// TIA Portal V17 export
// export: Created 2024-08-29T18:23:45.4451093Z, ExportSetting WithDefaults, DisplayName Totally Integrated Automation Portal, DisplayVersion V17 Update 7, DisplayName TIA Portal Openness, DisplayVersion V17 Update 7, DisplayName TIA Portal Version Control Interface, DisplayVersion V17, DisplayName SINAMICS Startdrive Advanced, DisplayVersion V17 SP2, DisplayName SINAMICS Startdrive G110M, G120, G120C, G120D, G120P, G115D, DisplayVersion V17 SP2, DisplayName SINAMICS Startdrive G130, G150, S120, S150, SINAMICS MV, S210, DisplayVersion V17 SP2, DisplayName STEP 7 Professional, DisplayVersion V17 Update 7, DisplayName STEP 7 Safety, DisplayVersion V17 Update 6, DisplayName WinCC Advanced / Unified PC, DisplayVersion V17 Update 7
FUNCTION "sensorStatus" : Void   // FC36, LAD
{ S7_Optimized_Access := 'TRUE' }
VERSION : 0.1
// stored: AutoNumber true, IsIECCheckEnabled false, SetENOAutomatically false, UDAEnableTagReadback false
   VAR_INPUT
      manualModeActive : Bool;
      automaticModeActive : Bool;
      sensorActive : Bool;
      sensorRequested : Bool;
      sensorMask : Bool;
   END_VAR
   VAR_OUTPUT
      sensorStatus : Int;
   END_VAR
   VAR_TEMP
      localMask : Bool;
   END_VAR
BEGIN

REGION Network 1
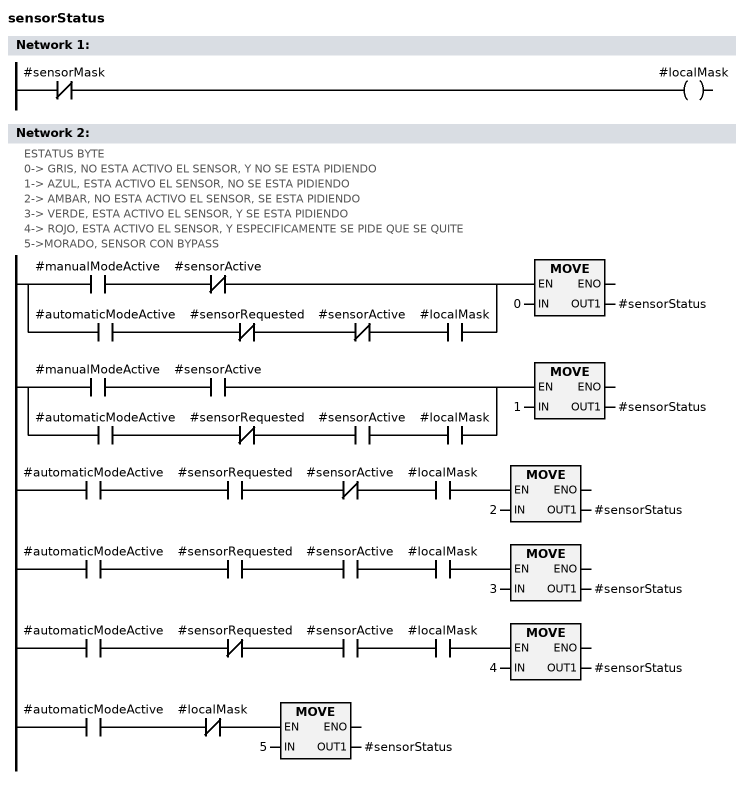
   RUNG wire#powerrail
      I_Contact( #sensorMask )
      Coil( #localMask )
   END_RUNG
   // the same network as SCL:
   #localMask := NOT #sensorMask;
END_REGION

REGION Network 2
   // ESTATUS BYTE
   // 0-> GRIS, NO ESTA ACTIVO EL SENSOR, Y NO SE ESTA PIDIENDO
   // 1-> AZUL, ESTA ACTIVO EL SENSOR, NO SE ESTA PIDIENDO
   // 2-> AMBAR, NO ESTA ACTIVO EL SENSOR, SE ESTA PIDIENDO
   // 3-> VERDE, ESTA ACTIVO EL SENSOR, Y SE ESTA PIDIENDO
   // 4-> ROJO, ESTA ACTIVO EL SENSOR, Y ESPECIFICAMENTE SE PIDE QUE SE QUITE
   // 5->MORADO, SENSOR CON BYPASS
   RUNG wire#powerrail
      Contact( #manualModeActive )
      I_Contact( #sensorActive )
      wire#w1
      Move(in := 0, out1 => #sensorStatus)
   END_RUNG
   RUNG wire#powerrail
      Contact( #automaticModeActive )
      I_Contact( #sensorRequested )
      I_Contact( #sensorActive )
      Contact( #localMask )
   END_RUNG wire#w1
   RUNG wire#powerrail
      Contact( #manualModeActive )
      Contact( #sensorActive )
      wire#w2
      Move(in := 1, out1 => #sensorStatus)
   END_RUNG
   RUNG wire#powerrail
      Contact( #automaticModeActive )
      I_Contact( #sensorRequested )
      Contact( #sensorActive )
      Contact( #localMask )
   END_RUNG wire#w2
   RUNG wire#powerrail
      Contact( #automaticModeActive )
      Contact( #sensorRequested )
      I_Contact( #sensorActive )
      Contact( #localMask )
      Move(in := 2, out1 => #sensorStatus)
   END_RUNG
   RUNG wire#powerrail
      Contact( #automaticModeActive )
      Contact( #sensorRequested )
      Contact( #sensorActive )
      Contact( #localMask )
      Move(in := 3, out1 => #sensorStatus)
   END_RUNG
   RUNG wire#powerrail
      Contact( #automaticModeActive )
      I_Contact( #sensorRequested )
      Contact( #sensorActive )
      Contact( #localMask )
      Move(in := 4, out1 => #sensorStatus)
   END_RUNG
   RUNG wire#powerrail
      Contact( #automaticModeActive )
      I_Contact( #localMask )
      Move(in := 5, out1 => #sensorStatus)
   END_RUNG
   // the same network as SCL:
   IF (#manualModeActive AND NOT #sensorActive) OR (#automaticModeActive AND NOT #sensorRequested AND NOT #sensorActive AND #localMask) THEN
       #sensorStatus := 0;
   END_IF;
   IF (#manualModeActive AND #sensorActive) OR (#automaticModeActive AND NOT #sensorRequested AND #sensorActive AND #localMask) THEN
       #sensorStatus := 1;
   END_IF;
   IF #automaticModeActive AND #sensorRequested AND NOT #sensorActive AND #localMask THEN
       #sensorStatus := 2;
   END_IF;
   IF #automaticModeActive AND #sensorRequested AND #sensorActive AND #localMask THEN
       #sensorStatus := 3;
   END_IF;
   IF #automaticModeActive AND NOT #sensorRequested AND #sensorActive AND #localMask THEN
       #sensorStatus := 4;
   END_IF;
   IF #automaticModeActive AND NOT #localMask THEN #sensorStatus := 5; END_IF;
END_REGION
END_FUNCTION
